Staubli VAL3: Rectangle3.dtx

public frame fReference = {x=1469.031, y=-405.47, z=-1108.651, rz=85.774, fatherId=world[0]}
public jointRx jPark = {j3=90, j5=90}
public jointRx jJoint = {j1=-33.26023, j2=80.10403, j3=50.99765, j5=48.89831, j6=-29.03404}
public mdesc mNomSpeed = {blend=off}
public mdesc mSpeed[9]
  [0] = {tmax=50, rmax=100, leave=0.1, reach=0.1, blend=cartesian}
  [1] = {tmax=50, rmax=100, leave=0.1, reach=0.1, blend=cartesian}
  [2] = {tmax=50, rmax=100, leave=0.1, reach=0.1, blend=cartesian}
  [3] = {tmax=50, rmax=100, leave=0.1, reach=0.1, blend=cartesian}
  [4] = {tmax=50, rmax=100, leave=0.1, reach=0.1, blend=cartesian}
  [5] = {tmax=50, rmax=100, leave=0.1, reach=0.1, blend=cartesian}
  [6] = {tmax=50, rmax=100, leave=0.1, reach=0.1, blend=cartesian}
  [7] = {tmax=50, rmax=100, leave=0.1, reach=0.1, blend=cartesian}
  [8] = {tmax=50, rmax=100, leave=0.1, reach=0.1, blend=cartesian}
public num nTraj
num nTimeStop
num nTimeStart
num nMode
num nEtat
public pointRx pPoint[306]
  [0] = {x=-572, y=-69, z=100, rx=180, rz=-90, shoulder=lefty, elbow=epositive, wrist=wpositive, fatherId=fReference[0]}
  [1] = {x=-572, y=-69, rx=180, rz=-90, shoulder=lefty, elbow=epositive, wrist=wpositive, fatherId=fReference[0]}
  [2] = {x=-572, y=-69, rx=180, rz=-90, shoulder=lefty, elbow=epositive, wrist=wpositive, fatherId=fReference[0]}
  [3] = {x=-572, y=-38.966, rx=180, rz=-90, shoulder=lefty, elbow=epositive, wrist=wpositive, fatherId=fReference[0]}
  [4] = {x=-572, y=-8.931, rx=180, rz=-90, shoulder=lefty, elbow=epositive, wrist=wpositive, fatherId=fReference[0]}
  [5] = {x=-572, y=21.103, rx=180, rz=-90, shoulder=lefty, elbow=epositive, wrist=wpositive, fatherId=fReference[0]}
  [6] = {x=-572, y=51.137, rx=180, rz=-89.077, shoulder=lefty, elbow=epositive, wrist=wpositive, fatherId=fReference[0]}
  [7] = {x=-571.516, y=81.159, rx=180, rz=-79.818, shoulder=lefty, elbow=epositive, wrist=wpositive, fatherId=fReference[0]}
  [8] = {x=-566.215, y=110.673, rx=180, rz=-68.571, shoulder=lefty, elbow=epositive, wrist=wpositive, fatherId=fReference[0]}
  [9] = {x=-555.26, y=138.586, rx=180, rz=-57.324, shoulder=lefty, elbow=epositive, wrist=wpositive, fatherId=fReference[0]}
  [10] = {x=-539.071, y=163.826, rx=180, rz=-46.076, shoulder=lefty, elbow=epositive, wrist=wpositive, fatherId=fReference[0]}
  [11] = {x=-518.27, y=185.424, rx=180, rz=-34.829, shoulder=lefty, elbow=epositive, wrist=wpositive, fatherId=fReference[0]}
  [12] = {x=-493.655, y=202.55, rx=180, rz=-23.582, shoulder=lefty, elbow=epositive, wrist=wpositive, fatherId=fReference[0]}
  [13] = {x=-466.173, y=214.546, rx=-180, rz=-12.334, shoulder=lefty, elbow=epositive, wrist=wpositive, fatherId=fReference[0]}
  [14] = {x=-436.879, y=220.952, rx=180, rz=-2.002, shoulder=lefty, elbow=epositive, wrist=wpositive, fatherId=fReference[0]}
  [15] = {x=-406.886, y=222, rx=180, shoulder=lefty, elbow=epositive, wrist=wpositive, fatherId=fReference[0]}
  [16] = {x=-376.852, y=222, rx=-180, shoulder=lefty, elbow=epositive, wrist=wpositive, fatherId=fReference[0]}
  [17] = {x=-346.817, y=222, rx=180, shoulder=lefty, elbow=epositive, wrist=wpositive, fatherId=fReference[0]}
  [18] = {x=-316.783, y=222, rx=180, shoulder=lefty, elbow=epositive, wrist=wpositive, fatherId=fReference[0]}
  [19] = {x=-286.749, y=222, rx=180, shoulder=lefty, elbow=epositive, wrist=wpositive, fatherId=fReference[0]}
  [20] = {x=-256.714, y=222, rx=180, shoulder=lefty, elbow=epositive, wrist=wpositive, fatherId=fReference[0]}
  [21] = {x=-226.68, y=222, rx=180, shoulder=lefty, elbow=epositive, wrist=wpositive, fatherId=fReference[0]}
  [22] = {x=-196.646, y=222, rx=-180, shoulder=lefty, elbow=epositive, wrist=wpositive, fatherId=fReference[0]}
  [23] = {x=-166.611, y=222, rx=180, shoulder=lefty, elbow=epositive, wrist=wpositive, fatherId=fReference[0]}
  [24] = {x=-136.577, y=222, rx=-180, shoulder=lefty, elbow=epositive, wrist=wpositive, fatherId=fReference[0]}
  [25] = {x=-106.543, y=222, rx=180, shoulder=lefty, elbow=epositive, wrist=wpositive, fatherId=fReference[0]}
  [26] = {x=-76.509, y=222, rx=180, shoulder=lefty, elbow=epositive, wrist=wpositive, fatherId=fReference[0]}
  [27] = {x=-46.474, y=222, rx=-180, shoulder=lefty, elbow=epositive, wrist=wpositive, fatherId=fReference[0]}
  [28] = {x=-16.44, y=222, rx=-180, shoulder=lefty, elbow=epositive, wrist=wpositive, fatherId=fReference[0]}
  [29] = {x=13.594, y=222, rx=-180, shoulder=lefty, elbow=epositive, wrist=wpositive, fatherId=fReference[0]}
  [30] = {x=43.629, y=222, rx=-180, shoulder=lefty, elbow=epositive, wrist=wpositive, fatherId=fReference[0]}
  [31] = {x=73.663, y=222, rx=180, shoulder=lefty, elbow=epositive, wrist=wpositive, fatherId=fReference[0]}
  [32] = {x=103.697, y=222, rx=180, shoulder=lefty, elbow=epositive, wrist=wpositive, fatherId=fReference[0]}
  [33] = {x=133.732, y=222, rx=180, shoulder=lefty, elbow=epositive, wrist=wpositive, fatherId=fReference[0]}
  [34] = {x=163.766, y=222, rx=-180, shoulder=lefty, elbow=epositive, wrist=wpositive, fatherId=fReference[0]}
  [35] = {x=193.8, y=222, rx=180, shoulder=lefty, elbow=epositive, wrist=wpositive, fatherId=fReference[0]}
  [36] = {x=223.834, y=222, rx=180, shoulder=lefty, elbow=epositive, wrist=wpositive, fatherId=fReference[0]}
  [37] = {x=253.869, y=222, rx=-180, shoulder=lefty, elbow=epositive, wrist=wpositive, fatherId=fReference[0]}
  [38] = {x=283.903, y=222, rx=-180, shoulder=lefty, elbow=epositive, wrist=wpositive, fatherId=fReference[0]}
  [39] = {x=313.937, y=222, rx=-180, shoulder=lefty, elbow=epositive, wrist=wpositive, fatherId=fReference[0]}
  [40] = {x=343.972, y=222, rx=-180, shoulder=lefty, elbow=epositive, wrist=wpositive, fatherId=fReference[0]}
  [41] = {x=374.006, y=222, rx=180, shoulder=lefty, elbow=epositive, wrist=wpositive, fatherId=fReference[0]}
  [42] = {x=404.04, y=222, rx=-180, rz=1.416, shoulder=lefty, elbow=epositive, wrist=wpositive, fatherId=fReference[0]}
  [43] = {x=434.05, y=221.258, rx=180, rz=11.269, shoulder=lefty, elbow=epositive, wrist=wpositive, fatherId=fReference[0]}
  [44] = {x=463.458, y=215.398, rx=-180, rz=22.516, shoulder=lefty, elbow=epositive, wrist=wpositive, fatherId=fReference[0]}
  [45] = {x=491.159, y=203.915, rx=-180, rz=33.763, shoulder=lefty, elbow=epositive, wrist=wpositive, fatherId=fReference[0]}
  [46] = {x=516.087, y=187.25, rx=180, rz=45.011, shoulder=lefty, elbow=epositive, wrist=wpositive, fatherId=fReference[0]}
  [47] = {x=537.287, y=166.043, rx=180, rz=56.258, shoulder=lefty, elbow=epositive, wrist=wpositive, fatherId=fReference[0]}
  [48] = {x=553.942, y=141.108, rx=-180, rz=67.505, shoulder=lefty, elbow=epositive, wrist=wpositive, fatherId=fReference[0]}
  [49] = {x=565.415, y=113.403, rx=-180, rz=78.753, shoulder=lefty, elbow=epositive, wrist=wpositive, fatherId=fReference[0]}
  [50] = {x=571.264, y=83.993, rx=-180, rz=88.594, shoulder=lefty, elbow=epositive, wrist=wpositive, fatherId=fReference[0]}
  [51] = {x=572, y=53.983, rx=-180, rz=90, shoulder=lefty, elbow=epositive, wrist=wpositive, fatherId=fReference[0]}
  [52] = {x=572, y=23.949, rx=-180, rz=90, shoulder=lefty, elbow=epositive, wrist=wpositive, fatherId=fReference[0]}
  [53] = {x=572, y=-6.086, rx=-180, rz=90, shoulder=lefty, elbow=epositive, wrist=wpositive, fatherId=fReference[0]}
  [54] = {x=572, y=-36.12, rx=-180, rz=90, shoulder=lefty, elbow=epositive, wrist=wpositive, fatherId=fReference[0]}
  [55] = {x=572, y=-66.154, rx=180, rz=94.608, shoulder=lefty, elbow=epositive, wrist=wpositive, fatherId=fReference[0]}
  [56] = {x=569.591, y=-96.046, rx=-180, rz=105.805, shoulder=lefty, elbow=epositive, wrist=wpositive, fatherId=fReference[0]}
  [57] = {x=561.423, y=-124.898, rx=180, rz=117.053, shoulder=lefty, elbow=epositive, wrist=wpositive, fatherId=fReference[0]}
  [58] = {x=547.785, y=-151.603, rx=180, rz=128.3, shoulder=lefty, elbow=epositive, wrist=wpositive, fatherId=fReference[0]}
  [59] = {x=529.201, y=-175.136, rx=180, rz=139.547, shoulder=lefty, elbow=epositive, wrist=wpositive, fatherId=fReference[0]}
  [60] = {x=506.383, y=-194.591, rx=-180, rz=150.795, shoulder=lefty, elbow=epositive, wrist=wpositive, fatherId=fReference[0]}
  [61] = {x=480.209, y=-209.223, rx=-180, rz=162.042, shoulder=lefty, elbow=epositive, wrist=wpositive, fatherId=fReference[0]}
  [62] = {x=451.684, y=-218.468, rx=-180, rz=173.289, shoulder=lefty, elbow=epositive, wrist=wpositive, fatherId=fReference[0]}
  [63] = {x=421.903, y=-221.972, rx=180, rz=174.947, shoulder=lefty, elbow=epositive, wrist=wpositive, fatherId=fReference[0]}
  [64] = {x=391.869, y=-222, rx=180, rz=176, shoulder=lefty, elbow=epositive, wrist=wpositive, fatherId=fReference[0]}
  [65] = {x=361.834, y=-222, rx=180, rz=177, shoulder=lefty, elbow=epositive, wrist=wpositive, fatherId=fReference[0]}
  [66] = {x=331.8, y=-222, rx=180, rz=178, shoulder=lefty, elbow=epositive, wrist=wpositive, fatherId=fReference[0]}
  [67] = {x=301.766, y=-222, rx=180, rz=179, shoulder=lefty, elbow=epositive, wrist=wpositive, fatherId=fReference[0]}
  [68] = {x=271.732, y=-222, rx=180, rz=180, shoulder=lefty, elbow=epositive, wrist=wpositive, fatherId=fReference[0]}
  [69] = {x=241.697, y=-222, rx=180, rz=180, shoulder=lefty, elbow=epositive, wrist=wpositive, fatherId=fReference[0]}
  [70] = {x=211.663, y=-222, rx=180, rz=180, shoulder=lefty, elbow=epositive, wrist=wpositive, fatherId=fReference[0]}
  [71] = {x=181.629, y=-222, rx=-180, rz=180, shoulder=lefty, elbow=epositive, wrist=wpositive, fatherId=fReference[0]}
  [72] = {x=151.594, y=-222, rx=180, rz=180, shoulder=lefty, elbow=epositive, wrist=wpositive, fatherId=fReference[0]}
  [73] = {x=121.56, y=-222, rx=180, rz=-180, shoulder=lefty, elbow=epositive, wrist=wpositive, fatherId=fReference[0]}
  [74] = {x=91.526, y=-222, rx=180, rz=180, shoulder=lefty, elbow=epositive, wrist=wpositive, fatherId=fReference[0]}
  [75] = {x=61.491, y=-222, rx=180, rz=180, shoulder=lefty, elbow=epositive, wrist=wpositive, fatherId=fReference[0]}
  [76] = {x=31.457, y=-222, rx=-180, rz=-180, shoulder=lefty, elbow=epositive, wrist=wpositive, fatherId=fReference[0]}
  [77] = {x=1.423, y=-222, rx=180, rz=180, shoulder=lefty, elbow=epositive, wrist=wpositive, fatherId=fReference[0]}
  [78] = {x=-28.611, y=-222, rx=180, rz=180, shoulder=lefty, elbow=epositive, wrist=wpositive, fatherId=fReference[0]}
  [79] = {x=-58.646, y=-222, rx=180, rz=180, shoulder=lefty, elbow=epositive, wrist=wpositive, fatherId=fReference[0]}
  [80] = {x=-88.68, y=-222, rx=-180, rz=180, shoulder=lefty, elbow=epositive, wrist=wpositive, fatherId=fReference[0]}
  [81] = {x=-118.714, y=-222, rx=-180, rz=180, shoulder=lefty, elbow=epositive, wrist=wpositive, fatherId=fReference[0]}
  [82] = {x=-148.749, y=-222, rx=180, rz=180, shoulder=lefty, elbow=epositive, wrist=wpositive, fatherId=fReference[0]}
  [83] = {x=-178.783, y=-222, rx=180, rz=180, shoulder=lefty, elbow=epositive, wrist=wpositive, fatherId=fReference[0]}
  [84] = {x=-208.817, y=-222, rx=180, rz=180, shoulder=lefty, elbow=epositive, wrist=wpositive, fatherId=fReference[0]}
  [85] = {x=-238.852, y=-222, rx=180, rz=180, shoulder=lefty, elbow=epositive, wrist=wpositive, fatherId=fReference[0]}
  [86] = {x=-268.886, y=-222, rx=180, rz=180, shoulder=lefty, elbow=epositive, wrist=wpositive, fatherId=fReference[0]}
  [87] = {x=-298.92, y=-222, rx=180, rz=180, shoulder=lefty, elbow=epositive, wrist=wpositive, fatherId=fReference[0]}
  [88] = {x=-328.954, y=-222, rx=180, rz=-180, shoulder=lefty, elbow=epositive, wrist=wpositive, fatherId=fReference[0]}
  [89] = {x=-358.989, y=-222, rx=180, rz=180, shoulder=lefty, elbow=epositive, wrist=wpositive, fatherId=fReference[0]}
  [90] = {x=-389.023, y=-222, rx=180, rz=-180, shoulder=lefty, elbow=epositive, wrist=wpositive, fatherId=fReference[0]}
  [91] = {x=-419.057, y=-222, rx=180, rz=-174.355, shoulder=lefty, elbow=epositive, wrist=wpositive, fatherId=fReference[0]}
  [92] = {x=-448.898, y=-219.05, rx=-180, rz=-163.108, shoulder=lefty, elbow=epositive, wrist=wpositive, fatherId=fReference[0]}
  [93] = {x=-477.59, y=-210.337, rx=180, rz=-155.86, shoulder=lefty, elbow=epositive, wrist=wpositive, fatherId=fReference[0]}
  [94] = {x=-504.032, y=-196.195, rx=180, rz=-155.613, shoulder=lefty, elbow=epositive, wrist=wpositive, fatherId=fReference[0]}
  [95] = {x=-527.208, y=-177.167, rx=180, rz=-154.366, shoulder=lefty, elbow=epositive, wrist=wpositive, fatherId=fReference[0]}
  [96] = {x=-546.227, y=-153.984, rx=-180, rz=-153.118, shoulder=lefty, elbow=epositive, wrist=wpositive, fatherId=fReference[0]}
  [97] = {x=-560.359, y=-127.537, rx=180, rz=-152.871, shoulder=lefty, elbow=epositive, wrist=wpositive, fatherId=fReference[0]}
  [98] = {x=-569.062, y=-98.842, rx=180, rz=-151.624, shoulder=lefty, elbow=epositive, wrist=wpositive, fatherId=fReference[0]}
  [99] = {x=-572, y=-69, rx=-180, rz=-151.624, shoulder=lefty, elbow=epositive, wrist=wpositive, fatherId=fReference[0]}
  [100] = {x=-572, y=-69, rx=-180, rz=-151.624, shoulder=lefty, elbow=epositive, wrist=wpositive, fatherId=fReference[0]}
  [101] = {x=-572, y=-69, z=100, rx=-180, rz=-151.624, shoulder=lefty, elbow=epositive, wrist=wpositive, fatherId=fReference[0]}
  [102] = {x=-572, y=-69, z=122, rx=180, rz=-151.624, shoulder=lefty, elbow=epositive, wrist=wpositive, fatherId=fReference[0]}
  [103] = {x=-572, y=-69, z=22, rx=-180, rz=-151.624, shoulder=lefty, elbow=epositive, wrist=wpositive, fatherId=fReference[0]}
  [104] = {x=-572, y=-69, z=22, rx=-180, rz=-151.624, shoulder=lefty, elbow=epositive, wrist=wpositive, fatherId=fReference[0]}
  [105] = {x=-569.062, y=-98.842, z=22, rx=180, rz=-151.871, shoulder=lefty, elbow=epositive, wrist=wpositive, fatherId=fReference[0]}
  [106] = {x=-560.359, y=-127.537, z=22, rx=180, rz=-153.118, shoulder=lefty, elbow=epositive, wrist=wpositive, fatherId=fReference[0]}
  [107] = {x=-546.227, y=-153.984, z=22, rx=180, rz=-153.366, shoulder=lefty, elbow=epositive, wrist=wpositive, fatherId=fReference[0]}
  [108] = {x=-527.208, y=-177.167, z=22, rx=180, rz=-154.613, shoulder=lefty, elbow=epositive, wrist=wpositive, fatherId=fReference[0]}
  [109] = {x=-504.032, y=-196.195, z=22, rx=180, rz=-154.86, shoulder=lefty, elbow=epositive, wrist=wpositive, fatherId=fReference[0]}
  [110] = {x=-477.59, y=-210.337, z=22, rx=180, rz=-163.108, shoulder=lefty, elbow=epositive, wrist=wpositive, fatherId=fReference[0]}
  [111] = {x=-448.898, y=-219.05, z=22, rx=180, rz=-174.355, shoulder=lefty, elbow=epositive, wrist=wpositive, fatherId=fReference[0]}
  [112] = {x=-419.057, y=-222, z=22, rx=180, rz=-180, shoulder=lefty, elbow=epositive, wrist=wpositive, fatherId=fReference[0]}
  [113] = {x=-389.023, y=-222, z=22, rx=180, rz=-180, shoulder=lefty, elbow=epositive, wrist=wpositive, fatherId=fReference[0]}
  [114] = {x=-358.989, y=-222, z=22, rx=180, rz=180, shoulder=lefty, elbow=epositive, wrist=wpositive, fatherId=fReference[0]}
  [115] = {x=-328.954, y=-222, z=22, rx=-180, rz=180, shoulder=lefty, elbow=epositive, wrist=wpositive, fatherId=fReference[0]}
  [116] = {x=-298.92, y=-222, z=22, rx=180, rz=180, shoulder=lefty, elbow=epositive, wrist=wpositive, fatherId=fReference[0]}
  [117] = {x=-268.886, y=-222, z=22, rx=-180, rz=180, shoulder=lefty, elbow=epositive, wrist=wpositive, fatherId=fReference[0]}
  [118] = {x=-238.852, y=-222, z=22, rx=180, rz=-180, shoulder=lefty, elbow=epositive, wrist=wpositive, fatherId=fReference[0]}
  [119] = {x=-208.817, y=-222, z=22, rx=180, rz=180, shoulder=lefty, elbow=epositive, wrist=wpositive, fatherId=fReference[0]}
  [120] = {x=-178.783, y=-222, z=22, rx=180, rz=180, shoulder=lefty, elbow=epositive, wrist=wpositive, fatherId=fReference[0]}
  [121] = {x=-148.749, y=-222, z=22, rx=-180, rz=180, shoulder=lefty, elbow=epositive, wrist=wpositive, fatherId=fReference[0]}
  [122] = {x=-118.714, y=-222, z=22, rx=-180, rz=180, shoulder=lefty, elbow=epositive, wrist=wpositive, fatherId=fReference[0]}
  [123] = {x=-88.68, y=-222, z=22, rx=180, rz=180, shoulder=lefty, elbow=epositive, wrist=wpositive, fatherId=fReference[0]}
  [124] = {x=-58.646, y=-222, z=22, rx=180, rz=180, shoulder=lefty, elbow=epositive, wrist=wpositive, fatherId=fReference[0]}
  [125] = {x=-28.611, y=-222, z=22, rx=180, rz=180, shoulder=lefty, elbow=epositive, wrist=wpositive, fatherId=fReference[0]}
  [126] = {x=1.423, y=-222, z=22, rx=180, rz=180, shoulder=lefty, elbow=epositive, wrist=wpositive, fatherId=fReference[0]}
  [127] = {x=31.457, y=-222, z=22, rx=180, rz=-180, shoulder=lefty, elbow=epositive, wrist=wpositive, fatherId=fReference[0]}
  [128] = {x=61.491, y=-222, z=22, rx=-180, rz=180, shoulder=lefty, elbow=epositive, wrist=wpositive, fatherId=fReference[0]}
  [129] = {x=91.526, y=-222, z=22, rx=180, rz=180, shoulder=lefty, elbow=epositive, wrist=wpositive, fatherId=fReference[0]}
  [130] = {x=121.56, y=-222, z=22, rx=-180, rz=-180, shoulder=lefty, elbow=epositive, wrist=wpositive, fatherId=fReference[0]}
  [131] = {x=151.594, y=-222, z=22, rx=-180, rz=180, shoulder=lefty, elbow=epositive, wrist=wpositive, fatherId=fReference[0]}
  [132] = {x=181.629, y=-222, z=22, rx=180, rz=180, shoulder=lefty, elbow=epositive, wrist=wpositive, fatherId=fReference[0]}
  [133] = {x=211.663, y=-222, z=22, rx=180, rz=180, shoulder=lefty, elbow=epositive, wrist=wpositive, fatherId=fReference[0]}
  [134] = {x=241.697, y=-222, z=22, rx=-180, rz=180, shoulder=lefty, elbow=epositive, wrist=wpositive, fatherId=fReference[0]}
  [135] = {x=271.732, y=-222, z=22, rx=180, rz=180, shoulder=lefty, elbow=epositive, wrist=wpositive, fatherId=fReference[0]}
  [136] = {x=301.766, y=-222, z=22, rx=-180, rz=179, shoulder=lefty, elbow=epositive, wrist=wpositive, fatherId=fReference[0]}
  [137] = {x=331.8, y=-222, z=22, rx=-180, rz=178, shoulder=lefty, elbow=epositive, wrist=wpositive, fatherId=fReference[0]}
  [138] = {x=361.834, y=-222, z=22, rx=180, rz=177, shoulder=lefty, elbow=epositive, wrist=wpositive, fatherId=fReference[0]}
  [139] = {x=391.869, y=-222, z=22, rx=180, rz=175.947, shoulder=lefty, elbow=epositive, wrist=wpositive, fatherId=fReference[0]}
  [140] = {x=421.903, y=-221.972, z=22, rx=180, rz=173.289, shoulder=lefty, elbow=epositive, wrist=wpositive, fatherId=fReference[0]}
  [141] = {x=451.684, y=-218.468, z=22, rx=180, rz=162.042, shoulder=lefty, elbow=epositive, wrist=wpositive, fatherId=fReference[0]}
  [142] = {x=480.209, y=-209.223, z=22, rx=180, rz=150.795, shoulder=lefty, elbow=epositive, wrist=wpositive, fatherId=fReference[0]}
  [143] = {x=506.383, y=-194.591, z=22, rx=180, rz=139.547, shoulder=lefty, elbow=epositive, wrist=wpositive, fatherId=fReference[0]}
  [144] = {x=529.201, y=-175.136, z=22, rx=-180, rz=128.3, shoulder=lefty, elbow=epositive, wrist=wpositive, fatherId=fReference[0]}
  [145] = {x=547.785, y=-151.603, z=22, rx=180, rz=117.053, shoulder=lefty, elbow=epositive, wrist=wpositive, fatherId=fReference[0]}
  [146] = {x=561.423, y=-124.898, z=22, rx=180, rz=105.805, shoulder=lefty, elbow=epositive, wrist=wpositive, fatherId=fReference[0]}
  [147] = {x=569.591, y=-96.046, z=22, rx=180, rz=94.608, shoulder=lefty, elbow=epositive, wrist=wpositive, fatherId=fReference[0]}
  [148] = {x=572, y=-66.154, z=22, rx=-180, rz=90, shoulder=lefty, elbow=epositive, wrist=wpositive, fatherId=fReference[0]}
  [149] = {x=572, y=-36.12, z=22, rx=-180, rz=90, shoulder=lefty, elbow=epositive, wrist=wpositive, fatherId=fReference[0]}
  [150] = {x=572, y=-6.086, z=22, rx=-180, rz=90, shoulder=lefty, elbow=epositive, wrist=wpositive, fatherId=fReference[0]}
  [151] = {x=572, y=23.949, z=22, rx=-180, rz=90, shoulder=lefty, elbow=epositive, wrist=wpositive, fatherId=fReference[0]}
  [152] = {x=572, y=53.983, z=22, rx=-180, rz=88.594, shoulder=lefty, elbow=epositive, wrist=wpositive, fatherId=fReference[0]}
  [153] = {x=571.264, y=83.993, z=22, rx=-180, rz=78.753, shoulder=lefty, elbow=epositive, wrist=wpositive, fatherId=fReference[0]}
  [154] = {x=565.415, y=113.403, z=22, rx=-180, rz=67.505, shoulder=lefty, elbow=epositive, wrist=wpositive, fatherId=fReference[0]}
  [155] = {x=553.942, y=141.108, z=22, rx=-180, rz=56.258, shoulder=lefty, elbow=epositive, wrist=wpositive, fatherId=fReference[0]}
  [156] = {x=537.287, y=166.043, z=22, rx=-180, rz=45.011, shoulder=lefty, elbow=epositive, wrist=wpositive, fatherId=fReference[0]}
  [157] = {x=516.087, y=187.25, z=22, rx=-180, rz=33.763, shoulder=lefty, elbow=epositive, wrist=wpositive, fatherId=fReference[0]}
  [158] = {x=491.159, y=203.915, z=22, rx=180, rz=22.516, shoulder=lefty, elbow=epositive, wrist=wpositive, fatherId=fReference[0]}
  [159] = {x=463.458, y=215.398, z=22, rx=-180, rz=11.269, shoulder=lefty, elbow=epositive, wrist=wpositive, fatherId=fReference[0]}
  [160] = {x=434.05, y=221.258, z=22, rx=-180, rz=1.416, shoulder=lefty, elbow=epositive, wrist=wpositive, fatherId=fReference[0]}
  [161] = {x=404.04, y=222, z=22, rx=-180, shoulder=lefty, elbow=epositive, wrist=wpositive, fatherId=fReference[0]}
  [162] = {x=374.006, y=222, z=22, rx=-180, shoulder=lefty, elbow=epositive, wrist=wpositive, fatherId=fReference[0]}
  [163] = {x=343.972, y=222, z=22, rx=180, shoulder=lefty, elbow=epositive, wrist=wpositive, fatherId=fReference[0]}
  [164] = {x=313.937, y=222, z=22, rx=180, shoulder=lefty, elbow=epositive, wrist=wpositive, fatherId=fReference[0]}
  [165] = {x=283.903, y=222, z=22, rx=180, shoulder=lefty, elbow=epositive, wrist=wpositive, fatherId=fReference[0]}
  [166] = {x=253.869, y=222, z=22, rx=-180, shoulder=lefty, elbow=epositive, wrist=wpositive, fatherId=fReference[0]}
  [167] = {x=223.834, y=222, z=22, rx=180, shoulder=lefty, elbow=epositive, wrist=wpositive, fatherId=fReference[0]}
  [168] = {x=193.8, y=222, z=22, rx=180, shoulder=lefty, elbow=epositive, wrist=wpositive, fatherId=fReference[0]}
  [169] = {x=163.766, y=222, z=22, rx=180, shoulder=lefty, elbow=epositive, wrist=wpositive, fatherId=fReference[0]}
  [170] = {x=133.732, y=222, z=22, rx=-180, shoulder=lefty, elbow=epositive, wrist=wpositive, fatherId=fReference[0]}
  [171] = {x=103.697, y=222, z=22, rx=180, shoulder=lefty, elbow=epositive, wrist=wpositive, fatherId=fReference[0]}
  [172] = {x=73.663, y=222, z=22, rx=-180, shoulder=lefty, elbow=epositive, wrist=wpositive, fatherId=fReference[0]}
  [173] = {x=43.629, y=222, z=22, rx=-180, shoulder=lefty, elbow=epositive, wrist=wpositive, fatherId=fReference[0]}
  [174] = {x=13.594, y=222, z=22, rx=180, shoulder=lefty, elbow=epositive, wrist=wpositive, fatherId=fReference[0]}
  [175] = {x=-16.44, y=222, z=22, rx=180, shoulder=lefty, elbow=epositive, wrist=wpositive, fatherId=fReference[0]}
  [176] = {x=-46.474, y=222, z=22, rx=180, shoulder=lefty, elbow=epositive, wrist=wpositive, fatherId=fReference[0]}
  [177] = {x=-76.509, y=222, z=22, rx=-180, shoulder=lefty, elbow=epositive, wrist=wpositive, fatherId=fReference[0]}
  [178] = {x=-106.543, y=222, z=22, rx=180, shoulder=lefty, elbow=epositive, wrist=wpositive, fatherId=fReference[0]}
  [179] = {x=-136.577, y=222, z=22, rx=-180, shoulder=lefty, elbow=epositive, wrist=wpositive, fatherId=fReference[0]}
  [180] = {x=-166.611, y=222, z=22, rx=-180, shoulder=lefty, elbow=epositive, wrist=wpositive, fatherId=fReference[0]}
  [181] = {x=-196.646, y=222, z=22, rx=-180, shoulder=lefty, elbow=epositive, wrist=wpositive, fatherId=fReference[0]}
  [182] = {x=-226.68, y=222, z=22, rx=180, shoulder=lefty, elbow=epositive, wrist=wpositive, fatherId=fReference[0]}
  [183] = {x=-256.714, y=222, z=22, rx=180, shoulder=lefty, elbow=epositive, wrist=wpositive, fatherId=fReference[0]}
  [184] = {x=-286.749, y=222, z=22, rx=180, shoulder=lefty, elbow=epositive, wrist=wpositive, fatherId=fReference[0]}
  [185] = {x=-316.783, y=222, z=22, rx=-180, shoulder=lefty, elbow=epositive, wrist=wpositive, fatherId=fReference[0]}
  [186] = {x=-346.817, y=222, z=22, rx=180, shoulder=lefty, elbow=epositive, wrist=wpositive, fatherId=fReference[0]}
  [187] = {x=-376.852, y=222, z=22, rx=180, shoulder=lefty, elbow=epositive, wrist=wpositive, fatherId=fReference[0]}
  [188] = {x=-406.886, y=222, z=22, rx=180, rz=-2.002, shoulder=lefty, elbow=epositive, wrist=wpositive, fatherId=fReference[0]}
  [189] = {x=-436.879, y=220.952, z=22, rx=180, rz=-12.334, shoulder=lefty, elbow=epositive, wrist=wpositive, fatherId=fReference[0]}
  [190] = {x=-466.173, y=214.546, z=22, rx=180, rz=-23.582, shoulder=lefty, elbow=epositive, wrist=wpositive, fatherId=fReference[0]}
  [191] = {x=-493.655, y=202.55, z=22, rx=180, rz=-34.829, shoulder=lefty, elbow=epositive, wrist=wpositive, fatherId=fReference[0]}
  [192] = {x=-518.27, y=185.424, z=22, rx=180, rz=-46.076, shoulder=lefty, elbow=epositive, wrist=wpositive, fatherId=fReference[0]}
  [193] = {x=-539.071, y=163.826, z=22, rx=180, rz=-57.324, shoulder=lefty, elbow=epositive, wrist=wpositive, fatherId=fReference[0]}
  [194] = {x=-555.26, y=138.586, z=22, rx=180, rz=-68.571, shoulder=lefty, elbow=epositive, wrist=wpositive, fatherId=fReference[0]}
  [195] = {x=-566.215, y=110.673, z=22, rx=180, rz=-79.818, shoulder=lefty, elbow=epositive, wrist=wpositive, fatherId=fReference[0]}
  [196] = {x=-571.516, y=81.159, z=22, rx=180, rz=-89.077, shoulder=lefty, elbow=epositive, wrist=wpositive, fatherId=fReference[0]}
  [197] = {x=-572, y=51.137, z=22, rx=180, rz=-90, shoulder=lefty, elbow=epositive, wrist=wpositive, fatherId=fReference[0]}
  [198] = {x=-572, y=21.103, z=22, rx=180, rz=-90, shoulder=lefty, elbow=epositive, wrist=wpositive, fatherId=fReference[0]}
  [199] = {x=-572, y=-8.931, z=22, rx=180, rz=-90, shoulder=lefty, elbow=epositive, wrist=wpositive, fatherId=fReference[0]}
  [200] = {x=-572, y=-38.966, z=22, rx=180, rz=-90, shoulder=lefty, elbow=epositive, wrist=wpositive, fatherId=fReference[0]}
  [201] = {x=-572, y=-69, z=22, rx=180, rz=-90, shoulder=lefty, elbow=epositive, wrist=wpositive, fatherId=fReference[0]}
  [202] = {x=-572, y=-69, z=22, rx=180, rz=-90, shoulder=lefty, elbow=epositive, wrist=wpositive, fatherId=fReference[0]}
  [203] = {x=-572, y=-69, z=122, rx=180, rz=-90, shoulder=lefty, elbow=epositive, wrist=wpositive, fatherId=fReference[0]}
  [204] = {x=-572, y=-69, z=144, rx=180, rz=-90, shoulder=lefty, elbow=epositive, wrist=wpositive, fatherId=fReference[0]}
  [205] = {x=-572, y=-69, z=44, rx=-180, rz=-90, shoulder=lefty, elbow=epositive, wrist=wpositive, fatherId=fReference[0]}
  [206] = {x=-572, y=-69, z=44, rx=-180, rz=-90, shoulder=lefty, elbow=epositive, wrist=wpositive, fatherId=fReference[0]}
  [207] = {x=-572, y=-38.966, z=44, rx=-180, rz=-90, shoulder=lefty, elbow=epositive, wrist=wpositive, fatherId=fReference[0]}
  [208] = {x=-572, y=-8.931, z=44, rx=180, rz=-90, shoulder=lefty, elbow=epositive, wrist=wpositive, fatherId=fReference[0]}
  [209] = {x=-572, y=21.103, z=44, rx=180, rz=-90, shoulder=lefty, elbow=epositive, wrist=wpositive, fatherId=fReference[0]}
  [210] = {x=-572, y=51.137, z=44, rx=180, rz=-89.077, shoulder=lefty, elbow=epositive, wrist=wpositive, fatherId=fReference[0]}
  [211] = {x=-571.516, y=81.159, z=44, rx=180, rz=-79.818, shoulder=lefty, elbow=epositive, wrist=wpositive, fatherId=fReference[0]}
  [212] = {x=-566.215, y=110.673, z=44, rx=180, rz=-68.571, shoulder=lefty, elbow=epositive, wrist=wpositive, fatherId=fReference[0]}
  [213] = {x=-555.26, y=138.586, z=44, rx=180, rz=-57.324, shoulder=lefty, elbow=epositive, wrist=wpositive, fatherId=fReference[0]}
  [214] = {x=-539.071, y=163.826, z=44, rx=180, rz=-46.076, shoulder=lefty, elbow=epositive, wrist=wpositive, fatherId=fReference[0]}
  [215] = {x=-518.27, y=185.424, z=44, rx=180, rz=-34.829, shoulder=lefty, elbow=epositive, wrist=wpositive, fatherId=fReference[0]}
  [216] = {x=-493.655, y=202.55, z=44, rx=180, rz=-23.582, shoulder=lefty, elbow=epositive, wrist=wpositive, fatherId=fReference[0]}
  [217] = {x=-466.173, y=214.546, z=44, rx=-180, rz=-12.334, shoulder=lefty, elbow=epositive, wrist=wpositive, fatherId=fReference[0]}
  [218] = {x=-436.879, y=220.952, z=44, rx=180, rz=-2.002, shoulder=lefty, elbow=epositive, wrist=wpositive, fatherId=fReference[0]}
  [219] = {x=-406.886, y=222, z=44, rx=-180, shoulder=lefty, elbow=epositive, wrist=wpositive, fatherId=fReference[0]}
  [220] = {x=-376.852, y=222, z=44, rx=180, shoulder=lefty, elbow=epositive, wrist=wpositive, fatherId=fReference[0]}
  [221] = {x=-346.817, y=222, z=44, rx=180, shoulder=lefty, elbow=epositive, wrist=wpositive, fatherId=fReference[0]}
  [222] = {x=-316.783, y=222, z=44, rx=180, shoulder=lefty, elbow=epositive, wrist=wpositive, fatherId=fReference[0]}
  [223] = {x=-286.749, y=222, z=44, rx=-180, shoulder=lefty, elbow=epositive, wrist=wpositive, fatherId=fReference[0]}
  [224] = {x=-256.714, y=222, z=44, rx=180, shoulder=lefty, elbow=epositive, wrist=wpositive, fatherId=fReference[0]}
  [225] = {x=-226.68, y=222, z=44, rx=-180, shoulder=lefty, elbow=epositive, wrist=wpositive, fatherId=fReference[0]}
  [226] = {x=-196.646, y=222, z=44, rx=-180, shoulder=lefty, elbow=epositive, wrist=wpositive, fatherId=fReference[0]}
  [227] = {x=-166.611, y=222, z=44, rx=-180, shoulder=lefty, elbow=epositive, wrist=wpositive, fatherId=fReference[0]}
  [228] = {x=-136.577, y=222, z=44, rx=180, shoulder=lefty, elbow=epositive, wrist=wpositive, fatherId=fReference[0]}
  [229] = {x=-106.543, y=222, z=44, rx=180, shoulder=lefty, elbow=epositive, wrist=wpositive, fatherId=fReference[0]}
  [230] = {x=-76.509, y=222, z=44, rx=-180, shoulder=lefty, elbow=epositive, wrist=wpositive, fatherId=fReference[0]}
  [231] = {x=-46.474, y=222, z=44, rx=180, shoulder=lefty, elbow=epositive, wrist=wpositive, fatherId=fReference[0]}
  [232] = {x=-16.44, y=222, z=44, rx=180, shoulder=lefty, elbow=epositive, wrist=wpositive, fatherId=fReference[0]}
  [233] = {x=13.594, y=222, z=44, rx=-180, shoulder=lefty, elbow=epositive, wrist=wpositive, fatherId=fReference[0]}
  [234] = {x=43.629, y=222, z=44, rx=-180, shoulder=lefty, elbow=epositive, wrist=wpositive, fatherId=fReference[0]}
  [235] = {x=73.663, y=222, z=44, rx=180, shoulder=lefty, elbow=epositive, wrist=wpositive, fatherId=fReference[0]}
  [236] = {x=103.697, y=222, z=44, rx=-180, shoulder=lefty, elbow=epositive, wrist=wpositive, fatherId=fReference[0]}
  [237] = {x=133.732, y=222, z=44, rx=180, shoulder=lefty, elbow=epositive, wrist=wpositive, fatherId=fReference[0]}
  [238] = {x=163.766, y=222, z=44, rx=-180, shoulder=lefty, elbow=epositive, wrist=wpositive, fatherId=fReference[0]}
  [239] = {x=193.8, y=222, z=44, rx=180, shoulder=lefty, elbow=epositive, wrist=wpositive, fatherId=fReference[0]}
  [240] = {x=223.834, y=222, z=44, rx=-180, shoulder=lefty, elbow=epositive, wrist=wpositive, fatherId=fReference[0]}
  [241] = {x=253.869, y=222, z=44, rx=-180, shoulder=lefty, elbow=epositive, wrist=wpositive, fatherId=fReference[0]}
  [242] = {x=283.903, y=222, z=44, rx=180, shoulder=lefty, elbow=epositive, wrist=wpositive, fatherId=fReference[0]}
  [243] = {x=313.937, y=222, z=44, rx=-180, shoulder=lefty, elbow=epositive, wrist=wpositive, fatherId=fReference[0]}
  [244] = {x=343.972, y=222, z=44, rx=-180, shoulder=lefty, elbow=epositive, wrist=wpositive, fatherId=fReference[0]}
  [245] = {x=374.006, y=222, z=44, rx=180, shoulder=lefty, elbow=epositive, wrist=wpositive, fatherId=fReference[0]}
  [246] = {x=404.04, y=222, z=44, rx=180, rz=1.416, shoulder=lefty, elbow=epositive, wrist=wpositive, fatherId=fReference[0]}
  [247] = {x=434.05, y=221.258, z=44, rx=-180, rz=11.269, shoulder=lefty, elbow=epositive, wrist=wpositive, fatherId=fReference[0]}
  [248] = {x=463.458, y=215.398, z=44, rx=-180, rz=22.516, shoulder=lefty, elbow=epositive, wrist=wpositive, fatherId=fReference[0]}
  [249] = {x=491.159, y=203.915, z=44, rx=-180, rz=33.763, shoulder=lefty, elbow=epositive, wrist=wpositive, fatherId=fReference[0]}
  [250] = {x=516.087, y=187.25, z=44, rx=180, rz=45.011, shoulder=lefty, elbow=epositive, wrist=wpositive, fatherId=fReference[0]}
  [251] = {x=537.287, y=166.043, z=44, rx=-180, rz=56.258, shoulder=lefty, elbow=epositive, wrist=wpositive, fatherId=fReference[0]}
  [252] = {x=553.942, y=141.108, z=44, rx=-180, rz=67.505, shoulder=lefty, elbow=epositive, wrist=wpositive, fatherId=fReference[0]}
  [253] = {x=565.415, y=113.403, z=44, rx=-180, rz=78.753, shoulder=lefty, elbow=epositive, wrist=wpositive, fatherId=fReference[0]}
  [254] = {x=571.264, y=83.993, z=44, rx=-180, rz=88.594, shoulder=lefty, elbow=epositive, wrist=wpositive, fatherId=fReference[0]}
  [255] = {x=572, y=53.983, z=44, rx=-180, rz=90, shoulder=lefty, elbow=epositive, wrist=wpositive, fatherId=fReference[0]}
  [256] = {x=572, y=23.949, z=44, rx=-180, rz=90, shoulder=lefty, elbow=epositive, wrist=wpositive, fatherId=fReference[0]}
  [257] = {x=572, y=-6.086, z=44, rx=-180, rz=90, shoulder=lefty, elbow=epositive, wrist=wpositive, fatherId=fReference[0]}
  [258] = {x=572, y=-36.12, z=44, rx=-180, rz=90, shoulder=lefty, elbow=epositive, wrist=wpositive, fatherId=fReference[0]}
  [259] = {x=572, y=-66.154, z=44, rx=180, rz=94.608, shoulder=lefty, elbow=epositive, wrist=wpositive, fatherId=fReference[0]}
  [260] = {x=569.591, y=-96.046, z=44, rx=180, rz=105.805, shoulder=lefty, elbow=epositive, wrist=wpositive, fatherId=fReference[0]}
  [261] = {x=561.423, y=-124.898, z=44, rx=180, rz=117.053, shoulder=lefty, elbow=epositive, wrist=wpositive, fatherId=fReference[0]}
  [262] = {x=547.785, y=-151.603, z=44, rx=-180, rz=128.3, shoulder=lefty, elbow=epositive, wrist=wpositive, fatherId=fReference[0]}
  [263] = {x=529.201, y=-175.136, z=44, rx=180, rz=139.547, shoulder=lefty, elbow=epositive, wrist=wpositive, fatherId=fReference[0]}
  [264] = {x=506.383, y=-194.591, z=44, rx=180, rz=150.795, shoulder=lefty, elbow=epositive, wrist=wpositive, fatherId=fReference[0]}
  [265] = {x=480.209, y=-209.223, z=44, rx=180, rz=162.042, shoulder=lefty, elbow=epositive, wrist=wpositive, fatherId=fReference[0]}
  [266] = {x=451.684, y=-218.468, z=44, rx=180, rz=173.289, shoulder=lefty, elbow=epositive, wrist=wpositive, fatherId=fReference[0]}
  [267] = {x=421.903, y=-221.972, z=44, rx=180, rz=174.947, shoulder=lefty, elbow=epositive, wrist=wpositive, fatherId=fReference[0]}
  [268] = {x=391.869, y=-222, z=44, rx=180, rz=176, shoulder=lefty, elbow=epositive, wrist=wpositive, fatherId=fReference[0]}
  [269] = {x=361.834, y=-222, z=44, rx=-180, rz=177, shoulder=lefty, elbow=epositive, wrist=wpositive, fatherId=fReference[0]}
  [270] = {x=331.8, y=-222, z=44, rx=180, rz=178, shoulder=lefty, elbow=epositive, wrist=wpositive, fatherId=fReference[0]}
  [271] = {x=301.766, y=-222, z=44, rx=-180, rz=179, shoulder=lefty, elbow=epositive, wrist=wpositive, fatherId=fReference[0]}
  [272] = {x=271.732, y=-222, z=44, rx=-180, rz=180, shoulder=lefty, elbow=epositive, wrist=wpositive, fatherId=fReference[0]}
  [273] = {x=241.697, y=-222, z=44, rx=180, rz=180, shoulder=lefty, elbow=epositive, wrist=wpositive, fatherId=fReference[0]}
  [274] = {x=211.663, y=-222, z=44, rx=180, rz=180, shoulder=lefty, elbow=epositive, wrist=wpositive, fatherId=fReference[0]}
  [275] = {x=181.629, y=-222, z=44, rx=180, rz=180, shoulder=lefty, elbow=epositive, wrist=wpositive, fatherId=fReference[0]}
  [276] = {x=151.594, y=-222, z=44, rx=180, rz=180, shoulder=lefty, elbow=epositive, wrist=wpositive, fatherId=fReference[0]}
  [277] = {x=121.56, y=-222, z=44, rx=-180, rz=-180, shoulder=lefty, elbow=epositive, wrist=wpositive, fatherId=fReference[0]}
  [278] = {x=91.526, y=-222, z=44, rx=180, rz=180, shoulder=lefty, elbow=epositive, wrist=wpositive, fatherId=fReference[0]}
  [279] = {x=61.491, y=-222, z=44, rx=-180, rz=180, shoulder=lefty, elbow=epositive, wrist=wpositive, fatherId=fReference[0]}
  [280] = {x=31.457, y=-222, z=44, rx=-180, rz=-180, shoulder=lefty, elbow=epositive, wrist=wpositive, fatherId=fReference[0]}
  [281] = {x=1.423, y=-222, z=44, rx=180, rz=180, shoulder=lefty, elbow=epositive, wrist=wpositive, fatherId=fReference[0]}
  [282] = {x=-28.611, y=-222, z=44, rx=180, rz=-180, shoulder=lefty, elbow=epositive, wrist=wpositive, fatherId=fReference[0]}
  [283] = {x=-58.646, y=-222, z=44, rx=-180, rz=180, shoulder=lefty, elbow=epositive, wrist=wpositive, fatherId=fReference[0]}
  [284] = {x=-88.68, y=-222, z=44, rx=-180, rz=180, shoulder=lefty, elbow=epositive, wrist=wpositive, fatherId=fReference[0]}
  [285] = {x=-118.714, y=-222, z=44, rx=-180, rz=-180, shoulder=lefty, elbow=epositive, wrist=wpositive, fatherId=fReference[0]}
  [286] = {x=-148.749, y=-222, z=44, rx=-180, rz=180, shoulder=lefty, elbow=epositive, wrist=wpositive, fatherId=fReference[0]}
  [287] = {x=-178.783, y=-222, z=44, rx=180, rz=180, shoulder=lefty, elbow=epositive, wrist=wpositive, fatherId=fReference[0]}
  [288] = {x=-208.817, y=-222, z=44, rx=180, rz=180, shoulder=lefty, elbow=epositive, wrist=wpositive, fatherId=fReference[0]}
  [289] = {x=-238.852, y=-222, z=44, rx=180, rz=-180, shoulder=lefty, elbow=epositive, wrist=wpositive, fatherId=fReference[0]}
  [290] = {x=-268.886, y=-222, z=44, rx=-180, rz=180, shoulder=lefty, elbow=epositive, wrist=wpositive, fatherId=fReference[0]}
  [291] = {x=-298.92, y=-222, z=44, rx=180, rz=180, shoulder=lefty, elbow=epositive, wrist=wpositive, fatherId=fReference[0]}
  [292] = {x=-328.954, y=-222, z=44, rx=-180, rz=180, shoulder=lefty, elbow=epositive, wrist=wpositive, fatherId=fReference[0]}
  [293] = {x=-358.989, y=-222, z=44, rx=180, rz=180, shoulder=lefty, elbow=epositive, wrist=wpositive, fatherId=fReference[0]}
  [294] = {x=-389.023, y=-222, z=44, rx=180, rz=-180, shoulder=lefty, elbow=epositive, wrist=wpositive, fatherId=fReference[0]}
  [295] = {x=-419.057, y=-222, z=44, rx=-180, rz=-174.355, shoulder=lefty, elbow=epositive, wrist=wpositive, fatherId=fReference[0]}
  [296] = {x=-448.898, y=-219.05, z=44, rx=180, rz=-163.108, shoulder=lefty, elbow=epositive, wrist=wpositive, fatherId=fReference[0]}
  [297] = {x=-477.59, y=-210.337, z=44, rx=180, rz=-155.86, shoulder=lefty, elbow=epositive, wrist=wpositive, fatherId=fReference[0]}
  [298] = {x=-504.032, y=-196.195, z=44, rx=-180, rz=-155.613, shoulder=lefty, elbow=epositive, wrist=wpositive, fatherId=fReference[0]}
  [299] = {x=-527.208, y=-177.167, z=44, rx=180, rz=-154.366, shoulder=lefty, elbow=epositive, wrist=wpositive, fatherId=fReference[0]}
  [300] = {x=-546.227, y=-153.984, z=44, rx=180, rz=-153.118, shoulder=lefty, elbow=epositive, wrist=wpositive, fatherId=fReference[0]}
  [301] = {x=-560.359, y=-127.537, z=44, rx=180, rz=-152.871, shoulder=lefty, elbow=epositive, wrist=wpositive, fatherId=fReference[0]}
  [302] = {x=-569.062, y=-98.842, z=44, rx=-180, rz=-151.624, shoulder=lefty, elbow=epositive, wrist=wpositive, fatherId=fReference[0]}
  [303] = {x=-572, y=-69, z=44, rx=180, rz=-151.624, shoulder=lefty, elbow=epositive, wrist=wpositive, fatherId=fReference[0]}
  [304] = {x=-572, y=-69, z=44, rx=180, rz=-151.624, shoulder=lefty, elbow=epositive, wrist=wpositive, fatherId=fReference[0]}
  [305] = {x=-572, y=-69, z=144, rx=180, rz=-151.624, shoulder=lefty, elbow=epositive, wrist=wpositive, fatherId=fReference[0]}
public tool tTool = {z=452, fatherId=flange[0], ioLink=valve1}
dio doPompe = {link=CanIO\RemIO\remio0_Q}
dio doPompe1 = {link=CanIO\RemIO\remio0_Q}
dio doValve1 = {link=valve1}
dio doValve2 = {link=valve2}
aio Tpompe = {link=CanIO\RemIO\remio0_QW}
aio Tpompe1 = {link=CanIO\RemIO\remio0_QW}
aio Tpompe2 = {link=CanIO\RemIO\remio0_QW}
num nTension = 1.2
num nTObtOpen = 2
num nTPompeOff = 2
num nTPompeOn = 2
